FUNCTION TryConvert_UDINT_TO_TIME : BOOL
VAR_INPUT
	in : UDINT;
	out : REFERENCE TO TIME;
END_VAR

out := UDINT_TO_TIME(in);
TryConvert_UDINT_TO_TIME := TRUE;

END_FUNCTION

(* stored: Version 1.1.0.1, ProductVersion 3.1.4024.12
   POU TryConvert_UDINT_TO_TIME: Id {0d8b0936-32e7-4cd5-a4fc-fa18c083a7db}, SpecialFunc None *)
